// Mitsubishi GX Works2 project: group_4_save_newlll   PLC: FX3G

// global labels: Global1
VAR_GLOBAL
  switch_start AT X010 : BOOL;
  lamp_day_work AT Y010 : BOOL;
  lamp_switch_day_work AT Y010 : BOOL;
  switch_check_start AT X010 : BOOL;
  clemantine AT D1110 : REAL;
  pomela AT D1120 : REAL;
  pulse_x10 AT X010 : BOOL;
END_VAR
VAR_GLOBAL CONSTANT
  con_st : REAL := 0.5;
  con_st_0 : REAL;
END_VAR
VAR_GLOBAL
  all_check AT Y010 : BOOL;
  circle AT Y010 : BOOL;
  wash_start AT X002 : BOOL;
  lamp_3_sec AT Y005 : BOOL;
END_VAR
VAR_GLOBAL CONSTANT
  count_down : INT := 300;
  count_3_sec : INT := 300;
END_VAR
VAR_GLOBAL
  lamp_along_day AT Y010 : BOOL;
  TC200 AT TC200 : BOOL;
  counter AT TC200 : BOOL;
  switch_counter_end AT TC200 : BOOL;
  switch_lamp AT TS200 : BOOL;
  TS200 AT TC200 : BOOL;
  orange AT D1100 : REAL;
END_VAR
VAR_GLOBAL CONSTANT
  con_50 : REAL := 50;
  con_2 : REAL := 2;
END_VAR
VAR_GLOBAL
  wash_orange AT D1200 : REAL;
  wash_clemantine AT D1210 : REAL;
  wash_pomela AT D1220 : REAL;
  stam AT Y001 : BOOL;
  all_fruit_container AT D1300 : REAL;
  X1_collect AT X001 : BOOL;
  Y1_collect_lamp AT Y001 : BOOL;
  switch_squize AT X011 : BOOL;
END_VAR
VAR_GLOBAL CONSTANT
  count_2 : WORD := 2;
END_VAR
VAR_GLOBAL
  cc0_2_press AT CC0 : BOOL;
  switch_end_count AT CS0 : BOOL;
  juise_container AT D1310 : REAL;
  counter_sqiuze AT TC210 : BOOL;
END_VAR
VAR_GLOBAL CONSTANT
  squize_3_sec : INT := 300;
END_VAR
VAR_GLOBAL
  switch_timer_finish AT TS210 : BOOL;
  M0_lamp AT M0 : BOOL;
  Timer_lamp_1 AT TC215 : BOOL;
END_VAR
VAR_GLOBAL CONSTANT
  count_time_1 : INT := 50;
END_VAR
VAR_GLOBAL
  end_timer_1 AT TS215 : BOOL;
  lamp_1 AT Y002 : BOOL;
END_VAR
VAR_GLOBAL CONSTANT
  count_time_2 : INT := 50;
END_VAR
VAR_GLOBAL
  lamp_2 AT Y003 : BOOL;
  Timer_lamp_2 AT TC217 : BOOL;
  end_timer_2 AT TS217 : BOOL;
  M1_finish AT M1 : BOOL;
  sertj AT M2 : BOOL;
  M2_chec_con AT M2 : BOOL;
  switch_stop_lamp AT X007 : BOOL;
  Timer_lamp_end_day AT TC219 : BOOL;
  Timer_lamp_finsh AT TC213 : BOOL;
  M3_lamp AT M3 : BOOL;
  Timer_lamp_finsh_stop AT TS213 : BOOL;
  lamp_along_day_glamp AT Y010 : BOOL;
  lamp_along_day_glamp1 AT Y010 : BOOL;
  switch_quality_check AT X003 : BOOL;
END_VAR
VAR_GLOBAL CONSTANT
  input_ge1 : INT;
  input_ge5 : INT := 5;
END_VAR
VAR_GLOBAL
  m4_state AT M4 : BOOL;
  good_quality : REAL;
  good_quality_juice_container AT D1320 : REAL;
END_VAR
VAR_GLOBAL CONSTANT
  count_4 : WORD := 400;
END_VAR
VAR_GLOBAL
  timer_lamp_3 AT TC203 : BOOL;
  switch_lamp_3 AT TS203 : BOOL;
END_VAR
VAR_GLOBAL CONSTANT
  count_5 : WORD := 500;
END_VAR
VAR_GLOBAL
  lamp_3 AT Y004 : BOOL;
  lamp_check AT M5 : BOOL;
  counter_times AT CC2 : BOOL;
  counter_times_pulse AT CS2 : BOOL;
  trash_container AT D1400 : REAL;
  save_analog_output AT D8201 : REAL;
  M6_stop_light AT M6 : BOOL;
  switch_find_min AT X006 : BOOL;
  switch_modulo_check AT X006 : BOOL;
END_VAR
VAR_GLOBAL CONSTANT
  con_3 : INT := 3;
END_VAR
VAR_GLOBAL
  lamp_waste AT Y006 : BOOL;
END_VAR
VAR_GLOBAL CONSTANT
  con_st_0_int : INT;
END_VAR
VAR_GLOBAL
  new_iteration AT X002 : BOOL;
  check_con AT X010 : BOOL;
  reset AT X002 : BOOL;
  TC_205 AT TC205 : BOOL;
  TS_205 AT TS205 : BOOL;
  M_7 AT M7 : BOOL;
  TC_207 AT TC207 : BOOL;
  TS_207 AT TS207 : BOOL;
  M_8 AT M8 : BOOL;
  TC_1 AT TC1 : BOOL;
  TS_1 AT TS1 : BOOL;
END_VAR
VAR_GLOBAL CONSTANT
  count_time_2x : INT := 5;
  con_st_false : BOOL;
END_VAR
VAR_GLOBAL
  M_9 AT M9 : BOOL;
  lamp_along_day_M10 AT M10 : BOOL;
  analog_test AT D8281 : INT;
  M_11 AT M11 : BOOL;
END_VAR
VAR_GLOBAL CONSTANT
  True_bit : BOOL := TRUE;
  con_404 : REAL := 404.5;
END_VAR
VAR_GLOBAL
  analog_ans AT D8282 : INT;
END_VAR
VAR_GLOBAL CONSTANT
  zero : INT;
  con_405 : INT := 405;
END_VAR
VAR_GLOBAL
  M_12 AT M12 : BOOL;
  input_M12 AT M12 : BOOL;
END_VAR

// task Task_01 (event TRUE, interval 0, priority 31): POU_01

PROGRAM POU_01
(* structured ladder/FBD written out as ST: instructions are called as NAME(EN, inputs, outputs); _pN, _eN, _tN stand for wires *)
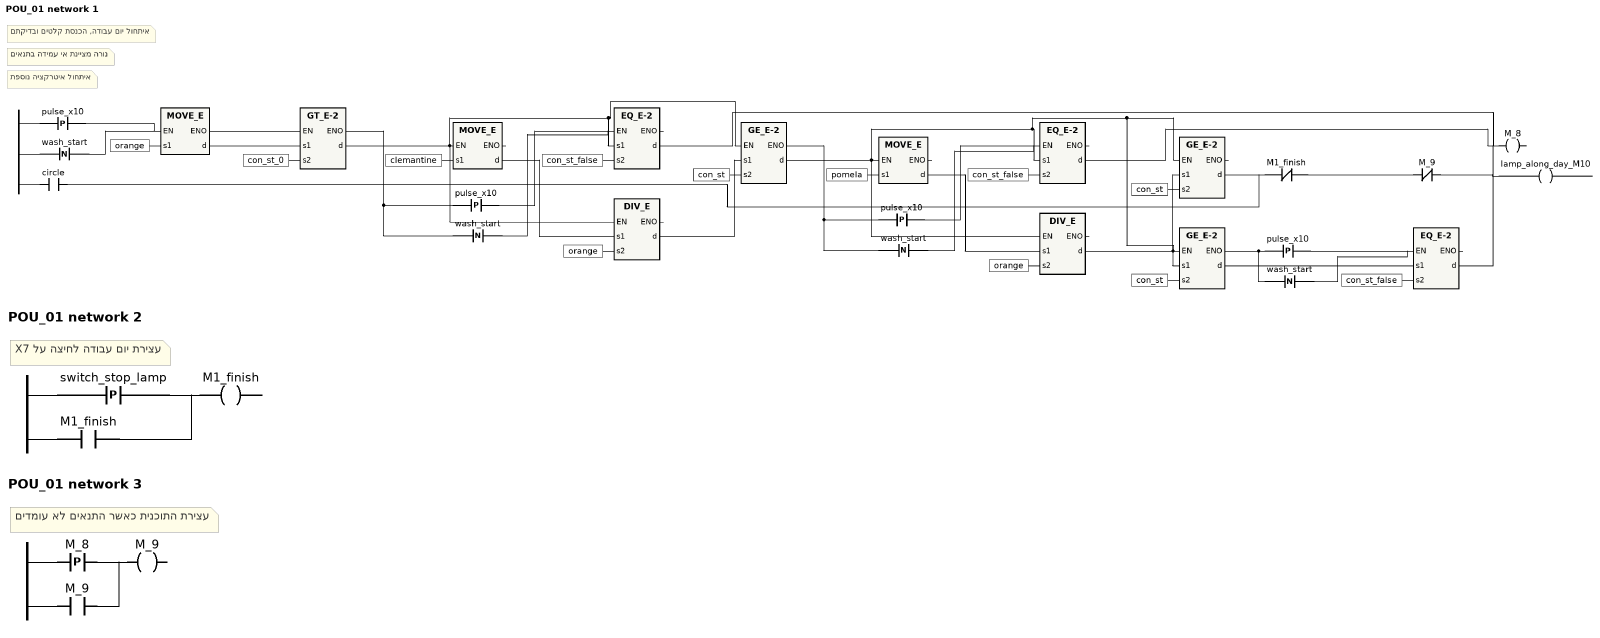
(* network 1 *)
(* איתחול יום עבודה, הכנסת קלטים ובדיקתם *)
(* נורה מציינת אי עמידה בתנאים *)
(* איתחול איטרקציה נוספת *)
_e2 := MOVE_E(LDP(TRUE, pulse_x10) OR LDF(TRUE, wash_start), orange, _t1);
_e4 := GT_E(_e2, _t1, con_st_0, _t3);
EQ_E((_e4 AND LDP(TRUE, pulse_x10)) OR (_e4 AND LDF(TRUE, wash_start)), _t3, con_st_false, _t5);
MOVE_E(_t3, clemantine, _t6);
DIV_E(_t3, _t6, orange, _t7);
_e9 := GE_E(_t3, _t7, con_st, _t8);
EQ_E((_e9 AND LDP(TRUE, pulse_x10)) OR (_e9 AND LDF(TRUE, wash_start)), _t8, con_st_false, _t10);
MOVE_E(_t8, pomela, _t11);
DIV_E(_t8, _t11, orange, _t12);
_e14 := GE_E(_t8, _t12, con_st, _t13);
EQ_E((_e14 AND LDP(TRUE, pulse_x10)) OR (_e14 AND LDF(TRUE, wash_start)), _t13, con_st_false, _t15);
M_8 := _t5 OR _t10 OR _t15;
GE_E(_t8, _t12, con_st, _t16);
lamp_along_day_M10 := ((_t16 OR circle) AND NOT M1_finish) AND NOT M_9;
(* network 2 *)
(* עצירת יום עבודה לחיצה על X7 *)
M1_finish := LDP(TRUE, switch_stop_lamp) OR M1_finish;
(* network 3 *)
(* עצירת התוכנית כאשר התנאים לא עומדים *)
M_9 := LDP(TRUE, M_8) OR M_9;
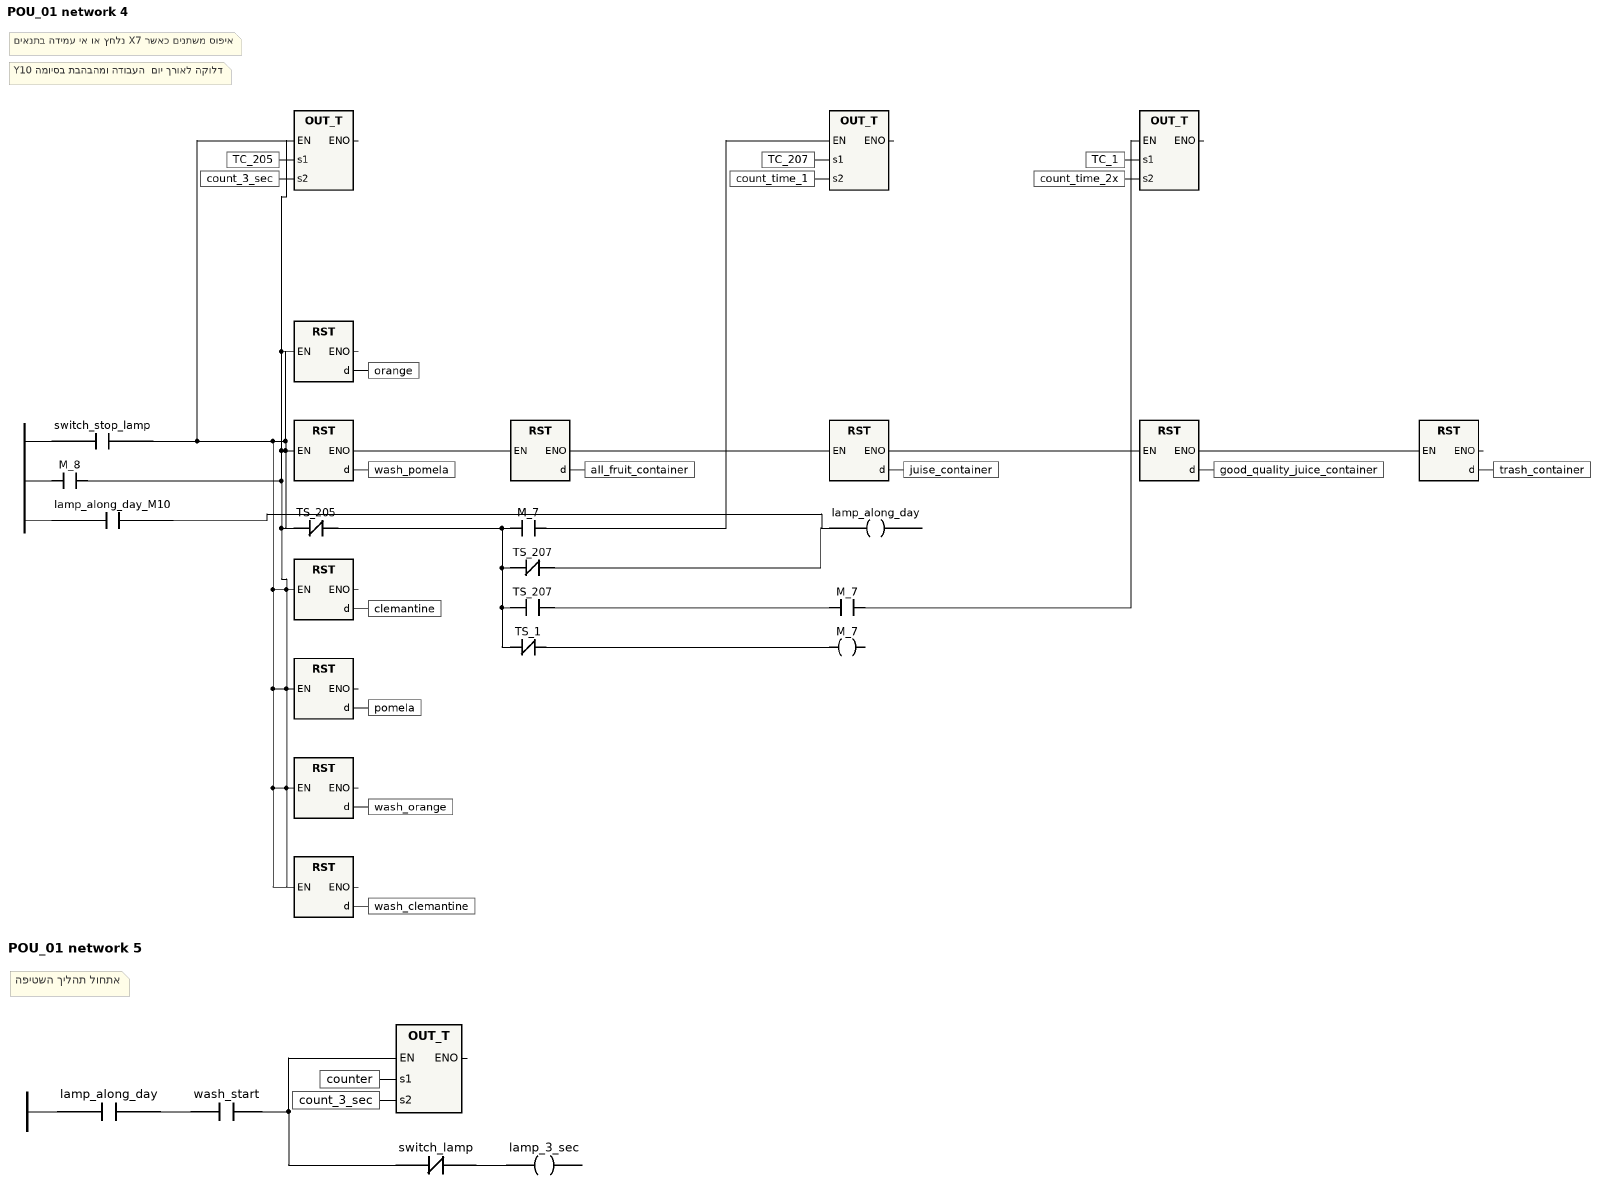
(* network 4 *)
(* איפוס משתנים כאשר X7 נלחץ או אי עמידה בתנאים *)
(* Y10 דלוקה לאורך יום  העבודה ומהבהבת בסיומה *)
_p1 := switch_stop_lamp OR M_8;
OUT_T(_p1, TC_205, count_3_sec);
_p2 := _p1 AND NOT TS_205;
OUT_T(_p2 AND M_7, TC_207, count_time_1);
RST(_p1, orange);
lamp_along_day := lamp_along_day_M10 OR (_p2 AND NOT TS_207);
RST(_p1, clemantine);
OUT_T(_p2 AND TS_207 AND M_7, TC_1, count_time_2x);
RST(_p1, pomela);
RST(_p1, wash_orange);
M_7 := _p2 AND NOT TS_1;
RST(_p1, wash_clemantine);
_e3 := RST(_p1, wash_pomela);
_e4 := RST(_e3, all_fruit_container);
_e5 := RST(_e4, juise_container);
_e6 := RST(_e5, good_quality_juice_container);
RST(_e6, trash_container);
(* network 5 *)
(* אתחול תהליך השטיפה *)
_p1 := lamp_along_day AND wash_start;
OUT_T(_p1, counter, count_3_sec);
lamp_3_sec := _p1 AND NOT switch_lamp;
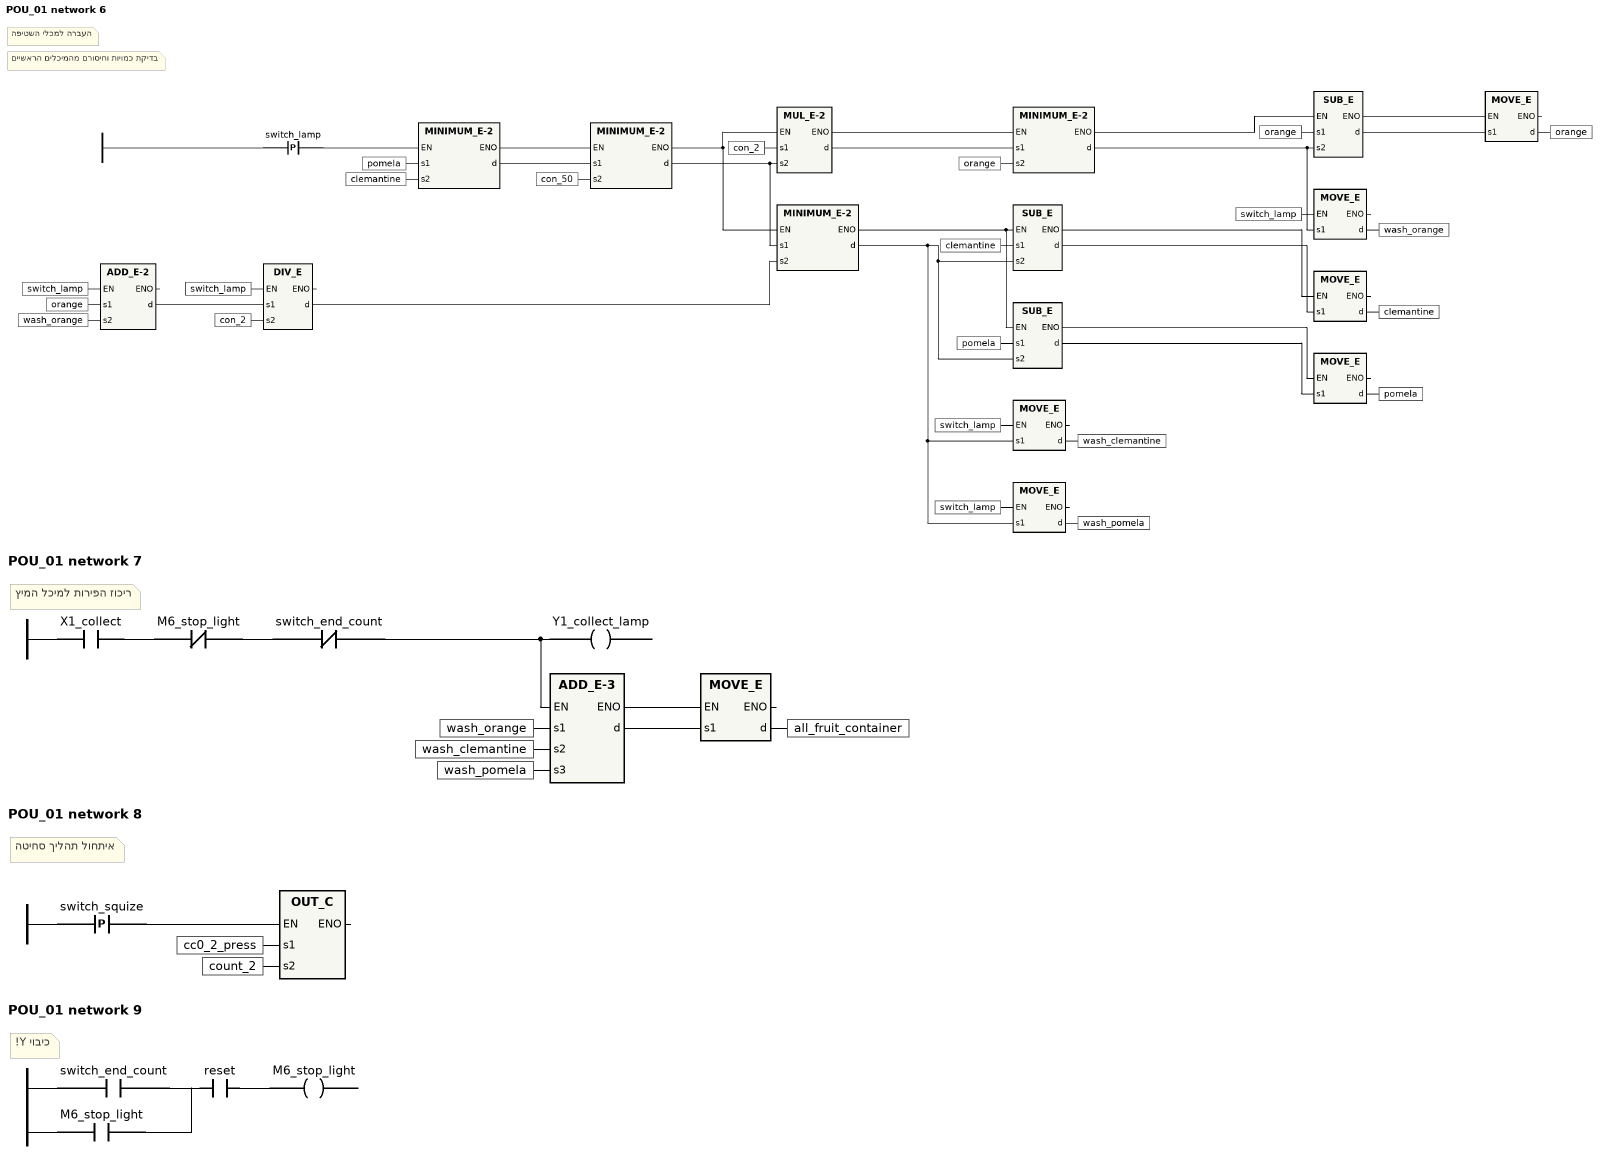
(* network 6 *)
(* העברה למכלי השטיפה *)
(* בדיקת כמויות וחיסורם מהמיכלים הראשיים *)
_e2 := MINIMUM_E(LDP(TRUE, switch_lamp), pomela, clemantine, _t1);
_e4 := MINIMUM_E(_e2, _t1, con_50, _t3);
_e6 := MUL_E(_e4, con_2, _t3, _t5);
_e8 := MINIMUM_E(_e6, _t5, orange, _t7);
_e10 := SUB_E(_e8, orange, _t7, _t9);
MOVE_E(_e10, _t9, orange);
MOVE_E(switch_lamp, _t7, wash_orange);
ADD_E(switch_lamp, orange, wash_orange, _t11);
DIV_E(switch_lamp, _t11, con_2, _t12);
_e14 := MINIMUM_E(_e4, _t3, _t12, _t13);
_e16 := SUB_E(_e14, clemantine, _t13, _t15);
MOVE_E(_e16, _t15, clemantine);
MOVE_E(switch_lamp, _t13, wash_clemantine);
MOVE_E(switch_lamp, _t13, wash_pomela);
_e18 := SUB_E(_e14, pomela, _t13, _t17);
MOVE_E(_e18, _t17, pomela);
(* network 7 *)
(* ריכוז הפירות למיכל המיץ *)
_p1 := X1_collect AND NOT M6_stop_light AND NOT switch_end_count;
Y1_collect_lamp := _p1;
_e3 := ADD_E(_p1, wash_orange, wash_clemantine, wash_pomela, _t2);
MOVE_E(_e3, _t2, all_fruit_container);
(* network 8 *)
(* איתחול תהליך סחיטה *)
OUT_C(LDP(TRUE, switch_squize), cc0_2_press, count_2);
(* network 9 *)
(* כיבוי Y! *)
M6_stop_light := (switch_end_count OR M6_stop_light) AND reset;
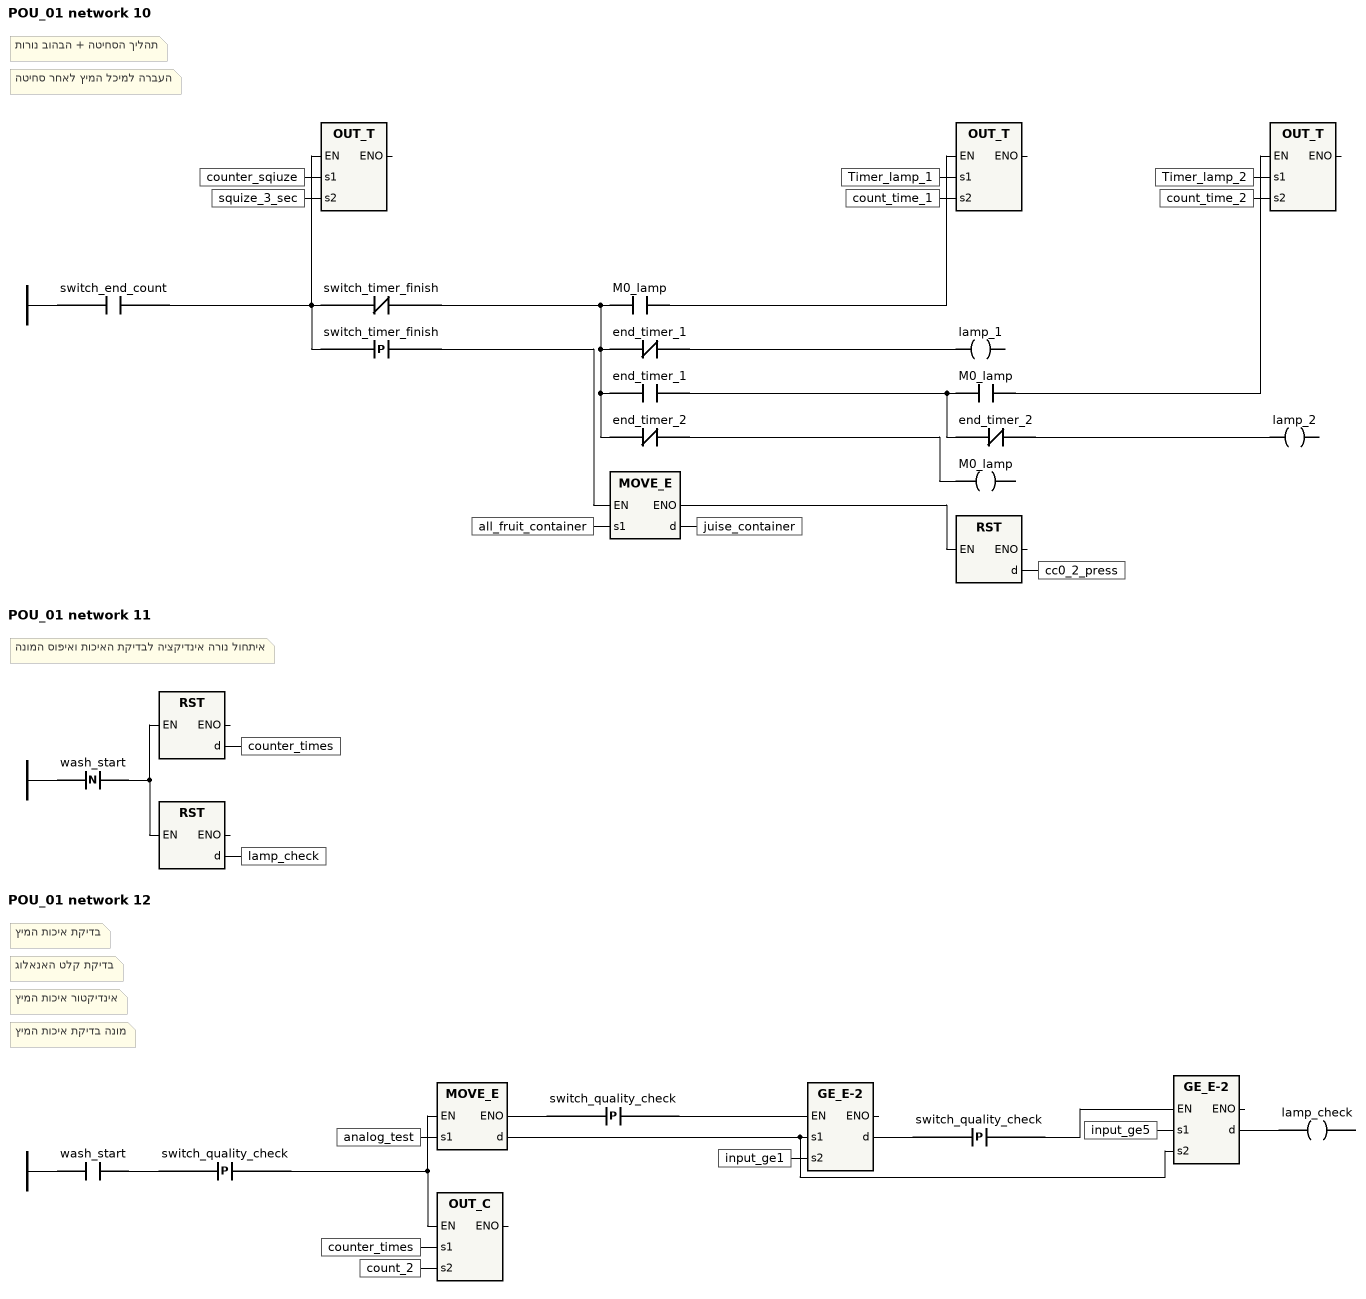
(* network 10 *)
(* תהליך הסחיטה + הבהוב נורות *)
(* העברה למיכל המיץ לאחר סחיטה *)
OUT_T(switch_end_count, counter_sqiuze, squize_3_sec);
_p1 := switch_end_count AND NOT switch_timer_finish;
OUT_T(_p1 AND M0_lamp, Timer_lamp_1, count_time_1);
lamp_1 := _p1 AND NOT end_timer_1;
_p2 := _p1 AND end_timer_1;
OUT_T(_p2 AND M0_lamp, Timer_lamp_2, count_time_2);
lamp_2 := _p2 AND NOT end_timer_2;
M0_lamp := _p1 AND NOT end_timer_2;
_e3 := MOVE_E(switch_end_count AND LDP(TRUE, switch_timer_finish), all_fruit_container, juise_container);
RST(_e3, cc0_2_press);
(* network 11 *)
(* איתחול נורה אינדיקציה לבדיקת האיכות ואיפוס המונה *)
_p1 := LDF(TRUE, wash_start);
RST(_p1, counter_times);
RST(_p1, lamp_check);
(* network 12 *)
(* בדיקת איכות המיץ *)
(* בדיקת קלט האנאלוג *)
(* אינדיקטור איכות המיץ *)
(* מונה בדיקת איכות המיץ *)
_p1 := wash_start AND LDP(TRUE, switch_quality_check);
_e3 := MOVE_E(_p1, analog_test, _t2);
GE_E(_e3 AND LDP(TRUE, switch_quality_check), _t2, input_ge1, _t4);
GE_E(_t4 AND LDP(TRUE, switch_quality_check), input_ge5, _t2, _t5);
lamp_check := _t5;
OUT_C(_p1, counter_times, count_2);
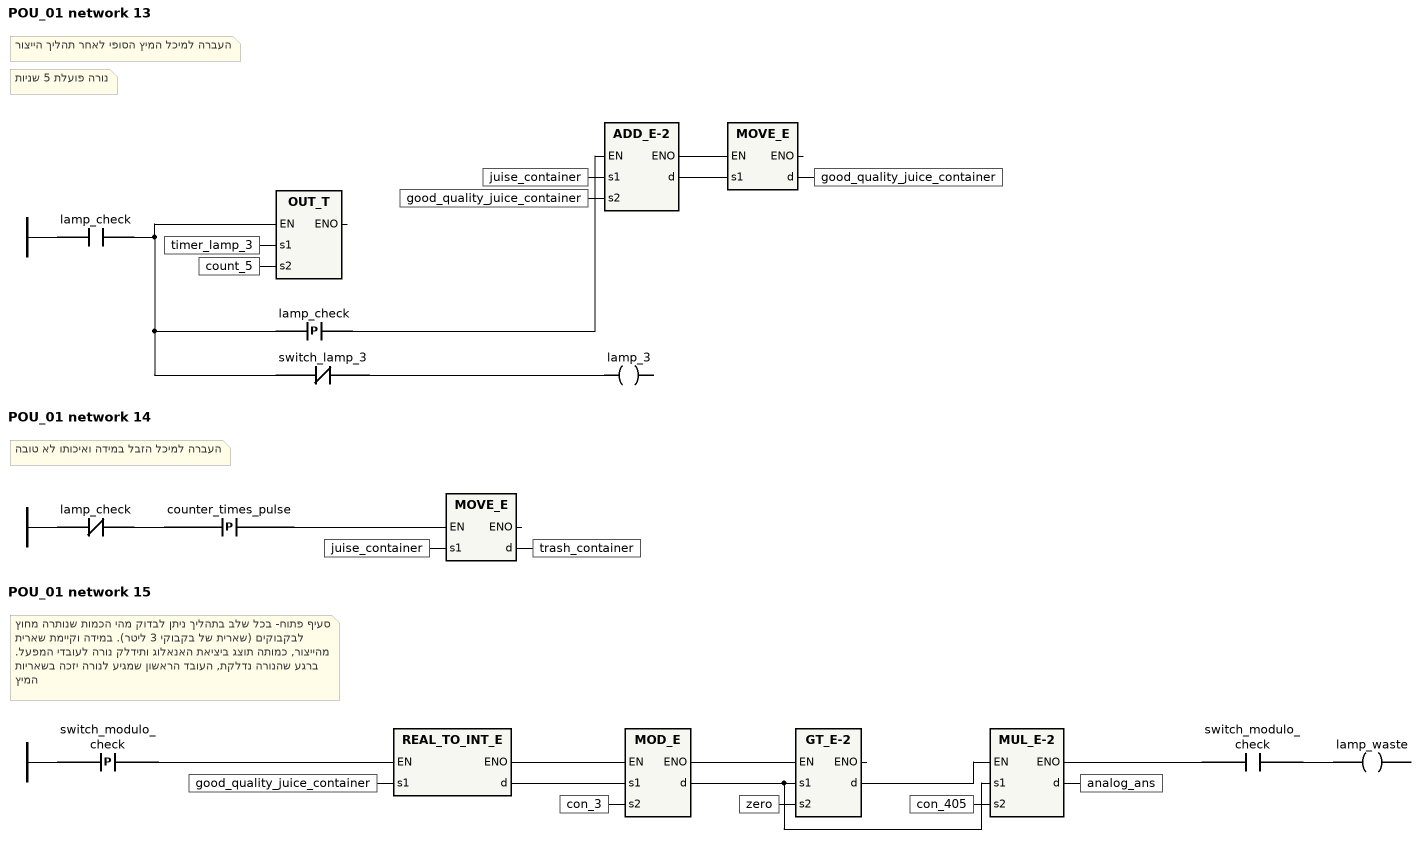
(* network 13 *)
(* העברה למיכל המיץ הסופי לאחר תהליך הייצור *)
(* נורה פועלת 5 שניות *)
_e2 := ADD_E(lamp_check AND LDP(TRUE, lamp_check), juise_container, good_quality_juice_container, _t1);
MOVE_E(_e2, _t1, good_quality_juice_container);
OUT_T(lamp_check, timer_lamp_3, count_5);
lamp_3 := lamp_check AND NOT switch_lamp_3;
(* network 14 *)
(* העברה למיכל הזבל במידה ואיכותו לא טובה *)
MOVE_E(NOT lamp_check AND LDP(TRUE, counter_times_pulse), juise_container, trash_container);
(* network 15 *)
(* סעיף פתוח- בכל שלב בתהליך ניתן לבדוק מהי הכמות שנותרה מחוץ לבקבוקים (שארית של בקבוקי 3 ליטר). במידה וקיימת שארית מהייצור, כמותה תוצג ביציאת האנאלוג ותידלק נורה לעובדי המפעל. ברגע שהנורה נדלקת, העובד הראשון שמגיע לנורה יזכה בשאריות המיץ *)
_e2 := REAL_TO_INT_E(LDP(TRUE, switch_modulo_check), good_quality_juice_container, _t1);
_e4 := MOD_E(_e2, _t1, con_3, _t3);
GT_E(_e4, _t3, zero, _t5);
_e6 := MUL_E(_t5, _t3, con_405, analog_ans);
lamp_waste := _e6 AND switch_modulo_check;
END_PROGRAM
